FUNCTION_BLOCK FB_PositionStateND
(*
    This function block coordinates multidimensional state moves for groups of motors.
    It is a building block not meant for use outside of lcls-twintcat-motion.

    Use FB_PositionState1D, FB_PositionState2D, ... etc. instead
*)
VAR_IN_OUT
    // Array of motors to move together
    astMotionStage: ARRAY[*] OF DUT_MotionStage;
    // 1D Position states: the current position to send each axis to
    astPositionState: ARRAY[*] OF DUT_PositionState;
    // 1D State movers: FBs to move the motors, need to be instantiated in the outer FB
    afbPositionStateMove: ARRAY[*] OF FB_PositionStateMove;
END_VAR
VAR_INPUT
    // Start all moves on rising edge, stop all moves on falling edge
    bExecute: BOOL;
    // Reset any errors
    bReset: BOOL;
    // Define behavior for when a move request is interrupted with a new request
    enumMotionRequest: ENUM_MotionRequest := ENUM_MotionRequest.WAIT;
END_VAR
VAR_OUTPUT
    // TRUE if ALL of the motors are at their goal states
    bAtState: BOOL;
    // TRUE if ANY of this FB's moves are in progress
    bBusy: BOOL;
    // TRUE if ALL motors have completed the last move request from this FB
    bDone: BOOL;
    // TRUE if ANY of this FB's moves had an error
    bError: BOOL;
    // How many FBs are erroring
    nErrorCount: UINT;
    // Which component is the source of the example/summarized error
    nShownError: DINT;
    // One of the error ids
    nErrorID: UDINT;
    // The error error message matching the ID
    sErrorMessage: STRING;
END_VAR
VAR
    nIndex: DINT;
    bInternalError: BOOL;
    nLowerBound: DINT;
    nUpperBound: DINT;
END_VAR


CheckArrayLengths();
IF NOT bInternalError THEN
    DoStateMoves();
    CombineOutputs();
END_IF

ACTION CheckArrayLengths:

// Get the bounds and make sure they are all the same
nLowerBound := LOWER_BOUND(astMotionStage, 1);
nUpperBound := UPPER_BOUND(astMotionStage, 1);

bInternalError S= nLowerBound <> LOWER_BOUND(astPositionState, 1);
bInternalError S= nUpperBound <> UPPER_BOUND(astPositionState, 1);
bInternalError S= nLowerBound <> LOWER_BOUND(afbPositionStateMove, 1);
bInternalError S= nUpperBound <> UPPER_BOUND(afbPositionStateMove, 1);

IF bInternalError THEN
    bError := TRUE;
    sErrorMessage := 'Internal Error: array lengths are inconsistent';
END_IF
END_ACTION

ACTION CombineOutputs:

// bAtState is TRUE if ALL entries are TRUE
bAtState := TRUE;
FOR nIndex := nLowerBound TO nUpperBound DO
    bAtState := bAtState AND afbPositionStateMove[nIndex].bAtState;
END_FOR

// bBusy is TRUE if ANY entry is TRUE
bBusy := FALSE;
FOR nIndex := nLowerBound TO nUpperBound DO
    bBusy := bBusy OR afbPositionStateMove[nIndex].bBusy;
END_FOR

// bDone is TRUE if ALL entries are TRUE
bDone := TRUE;
FOR nIndex := nLowerBound TO nUpperBound DO
    bDone := bDone AND afbPositionStateMove[nIndex].bDone;
END_FOR

// bError is TRUE if ANY entry is TRUE
// also set nShownError and increment nErrorCount
bError := FALSE;
nErrorCount := 0;
FOR nIndex := nLowerBound TO nUpperBound DO
    bError := bError OR afbPositionStateMove[nIndex].bError;
    IF afbPositionStateMove[nIndex].bError THEN
        nShownError := nIndex;
        nErrorCount := nErrorCount + 1;
    END_IF
END_FOR

// Pick error id and message using nShownError
IF bError THEN
    nErrorID := afbPositionStateMove[nShownError].nErrorID;
    sErrorMessage := afbPositionStateMove[nShownError].sErrorMessage;
ELSE
    nErrorID := 0;
    sErrorMessage := '';
END_IF
END_ACTION

ACTION DoStateMoves:

// Do the individual moves
FOR nIndex := nLowerBound TO nUpperBound DO
    afbPositionStateMove[nIndex](
        stMotionStage:=astMotionStage[nIndex],
        stPositionState:=astPositionState[nIndex],
        bExecute:=bExecute,
        bReset:=bReset,
        enumMotionRequest:=enumMotionRequest,
    );
END_FOR
END_ACTION

END_FUNCTION_BLOCK

(* stored: Version 1.1.0.1, ProductVersion 3.1.4022.18
   POU FB_PositionStateND: Id {27786e6e-dd37-418c-9b7c-370d3ce7e59f}, SpecialFunc None
   Action CheckArrayLengths: Id {9244b3c0-fac6-4a82-83fe-d3ec9dc81390}
   Action CombineOutputs: Id {fb280db4-19e3-45d0-a523-0567a14368b1}
   Action DoStateMoves: Id {d81e9830-b01d-4422-98b3-41033ba5b368} *)
